# EPICS substitutions: db/empty.substitutions
file empty.template
{
  pattern {}
}
